Omron Sysmac Studio project Colorificio_grafica_MK.3 (Sysmac Studio 1.30.0.17, StandardProject)

# Controller PLC: NX1P2-9024DT1 version 1.40
Task PrimaryTask (priority 4, period or condition 2000): Program0
Library OmronLib_WC_Toolbox_V1_0 1.0.0 (contents left out)

TYPE S_Colori : STRUCT
    ALPHA : INT;
    RED : INT;
    GREEN : INT;
    BLU : INT;
    NOME : STRING[256];
END_STRUCT END_TYPE

VAR_GLOBAL
    SB0 : BOOL;  (* pulsante avvio ciclo automatico *)
    SB1 : BOOL;  (* pulsante arresto ciclo automatico *)
    SBE : BOOL;  (* pulsante arresto di emergenza *)
    YVA : BOOL;  (* libera caricatore seconda latta (A-) *)
    YVB : BOOL;  (* libera caricatore prima latta (B-) *)
    YVC : BOOL;  (* scarico bilancia (C+) *)
    KM1 : BOOL;  (* motore primo nastro *)
    KM2 : BOOL;  (* motore secondo nastro *)
    YVD : BOOL;  (* scarico coperchiatrice (D+) *)
    a0 : BOOL := False;  (* caricatore seconda latta libero (NA) *)
    a1 : BOOL := True;  (* caricatore seconda latta bloccato (NA) *)
    b0 : BOOL := False;  (* caricatore prima latta libero (NA) *)
    b1 : BOOL := True;  (* caricatore prima latta bloccato (NA) *)
    c0 : BOOL := True;  (* scaricatore bilancia rientrato (NA) *)
    c1 : BOOL := False;  (* scaricatore bilancia esteso (NA) *)
    d0 : BOOL := True;  (* scaricatore coperchiatrice rientrato (NA) *)
    d1 : BOOL := False;  (* scaricatore coperchiatrice esteso (NA) *)
    BIL : REAL;  (* bilancia/cella di carico (Grammi) *)
    YVBASE : BOOL;  (* eroga colorante base *)
    YVRED : BOOL;  (* eroga colorante rosso *)
    YVGREEN : BOOL;  (* eroga colorante verde *)
    YVBLU : BOOL;  (* eroga colorante blu *)
    YVSCARICO : BOOL;  (* eroga totale colore *)
    Tbase : TIME;  (* tempo carico base *)
    Trosso : TIME;  (* tempo carico rosso *)
    Tgreen : TIME;  (* tempo carico verde *)
    Tblu : TIME;  (* tempo carico blu *)
    BLW0 : BOOL := True;  (* livello minimo Base White (NA) *)
    BLW1 : BOOL := True;  (* livello riserva Base White (NA) *)
    BLR0 : BOOL := True;  (* livello minimo Red (NA) *)
    BLR1 : BOOL := True;  (* livello riserva Red (NA) *)
    BLG0 : BOOL := True;  (* livello minimo Green (NA) *)
    BLG1 : BOOL := True;  (* livello riserva Green (NA) *)
    BLB0 : BOOL := True;  (* livello minimo Blu (NA) *)
    BLB1 : BOOL := True;  (* livello riserva Blu (NA) *)
    BC0 : BOOL := False;  (* presenza prima latta sul caricatore (NA) *)
    BC1 : BOOL := False;  (* presenza seconda latta sul caricatore (NA) *)
    BBIL : BOOL := False;  (* presenza sulla bilancia (NA) *)
    BCOP : BOOL := False;  (* presenza sulla coperchiatrice (NA) *)
    ContattoValvolaBase : BOOL;
    ContattoValvolaRosso : BOOL;
    ContattoValvolaVerde : BOOL;
    ContattoValvolaBlu : BOOL;
    ContattoValvolaTramoggia : BOOL;
    LevelToEjectBase : INT := -1;
    LevelToEjectRosso : INT := -1;
    LevelToEjectVerde : INT := -1;
    LevelToEjectBlu : INT := -1;
    ColorDone : BOOL := False;
END_VAR

PROGRAM Program0
VAR
    TimerBase : TP;
    TimerRosso : TP;
    TimerVerde : TP;
    TimerBlu : TP;
    estimatedBase : TIME;
    estimatedRosso : TIME;
    estimatedVerde : TIME;
    estimatedBlu : TIME;
    SeqRGB : BOOL;
    Base : BOOL;
    Rosso : BOOL;
    Verde : BOOL;
    Blu : BOOL;
END_VAR
VAR_EXTERNAL
    SB1 : BOOL;
    KM1 : BOOL;
    YVC : BOOL;
    BBIL : BOOL;
    c0 : BOOL;
    c1 : BOOL;
    KM2 : BOOL;
    SB0 : BOOL;
    SBE : BOOL;
    BIL : REAL;
    ContattoValvolaBase : BOOL;
    ContattoValvolaRosso : BOOL;
    ContattoValvolaVerde : BOOL;
    ContattoValvolaBlu : BOOL;
    YVBASE : BOOL;
    YVRED : BOOL;
    YVGREEN : BOOL;
    YVBLU : BOOL;
    Tbase : TIME;
    Trosso : TIME;
    Tgreen : TIME;
    Tblu : TIME;
    ContattoValvolaTramoggia : BOOL;
    YVSCARICO : BOOL;
    LevelToEjectBase : INT;
    LevelToEjectRosso : INT;
    LevelToEjectVerde : INT;
    LevelToEjectBlu : INT;
    ColorDone : BOOL;  (* Finito il processo di carica della latta *)
END_VAR
VAR
    _p1 : BOOL;
    _p2 : BOOL;
    _p3 : BOOL;
END_VAR

(* Section Section0: ladder, written here as Structured Text *)

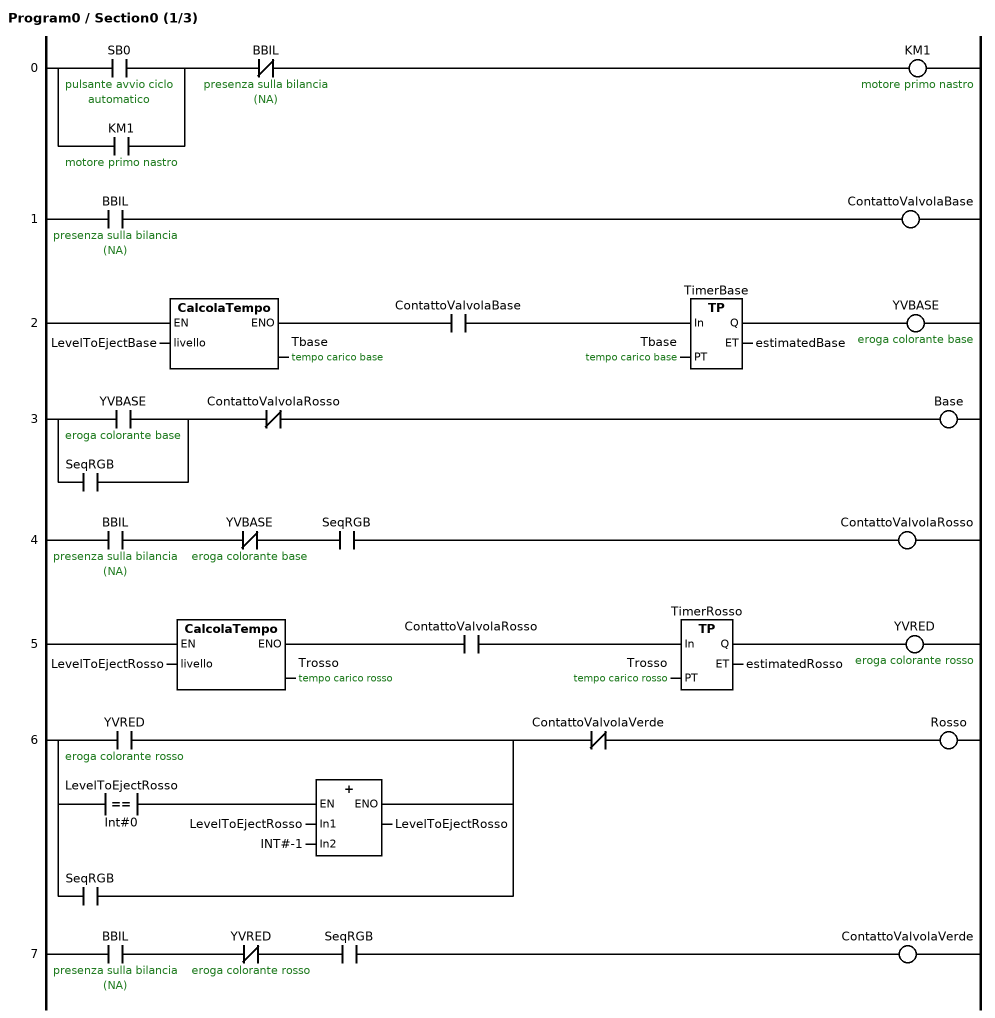
(* Rung 0 *)
KM1 := (SB0 OR KM1) AND NOT BBIL;
(* Rung 1 *)
ContattoValvolaBase := BBIL;
(* Rung 2 *)
Tbase := CalcolaTempo(livello := LevelToEjectBase);
TimerBase(In := ContattoValvolaBase, PT := Tbase, ET => estimatedBase);
YVBASE := TimerBase.Q;
(* Rung 3 *)
Base := (YVBASE OR SeqRGB) AND NOT ContattoValvolaRosso;
(* Rung 4 *)
ContattoValvolaRosso := BBIL AND NOT YVBASE AND SeqRGB;
(* Rung 5 *)
Trosso := CalcolaTempo(livello := LevelToEjectRosso);
TimerRosso(In := ContattoValvolaRosso, PT := Trosso, ET => estimatedRosso);
YVRED := TimerRosso.Q;
(* Rung 6 *)
_p1 := LevelToEjectRosso = Int#0;
IF _p1 THEN LevelToEjectRosso := LevelToEjectRosso + (INT#-1); END_IF;
Rosso := (YVRED OR _p1 OR SeqRGB) AND NOT ContattoValvolaVerde;
(* Rung 7 *)
ContattoValvolaVerde := BBIL AND NOT YVRED AND SeqRGB;

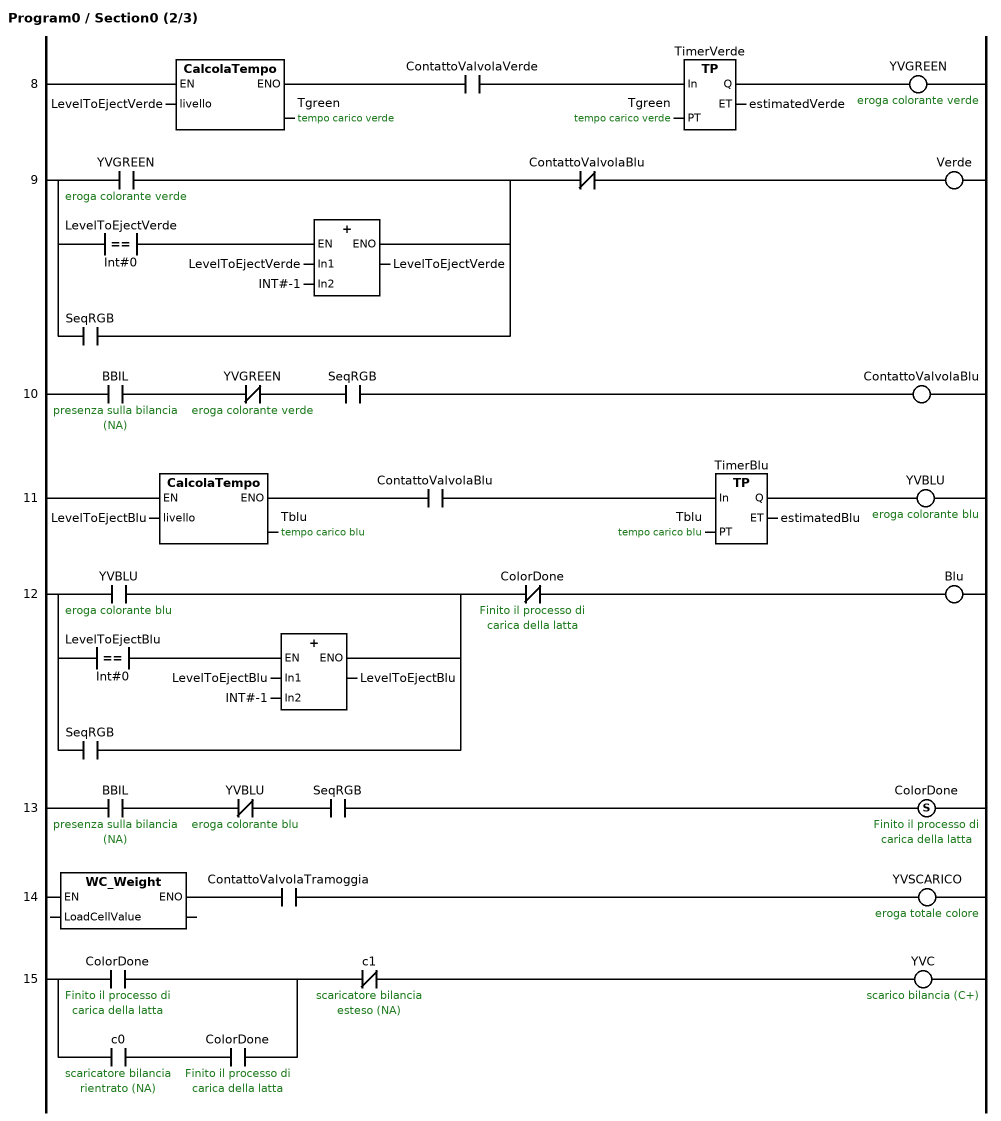
(* Rung 8 *)
Tgreen := CalcolaTempo(livello := LevelToEjectVerde);
TimerVerde(In := ContattoValvolaVerde, PT := Tgreen, ET => estimatedVerde);
YVGREEN := TimerVerde.Q;
(* Rung 9 *)
_p2 := LevelToEjectVerde = Int#0;
IF _p2 THEN LevelToEjectVerde := LevelToEjectVerde + (INT#-1); END_IF;
Verde := (YVGREEN OR _p2 OR SeqRGB) AND NOT ContattoValvolaBlu;
(* Rung 10 *)
ContattoValvolaBlu := BBIL AND NOT YVGREEN AND SeqRGB;
(* Rung 11 *)
Tblu := CalcolaTempo(livello := LevelToEjectBlu);
TimerBlu(In := ContattoValvolaBlu, PT := Tblu, ET => estimatedBlu);
YVBLU := TimerBlu.Q;
(* Rung 12 *)
_p3 := LevelToEjectBlu = Int#0;
IF _p3 THEN LevelToEjectBlu := LevelToEjectBlu + (INT#-1); END_IF;
Blu := (YVBLU OR _p3 OR SeqRGB) AND NOT ColorDone;
(* Rung 13 *)
IF BBIL AND NOT YVBLU AND SeqRGB THEN ColorDone := TRUE; END_IF;
(* Rung 14 *)
WC_Weight();
YVSCARICO := ContattoValvolaTramoggia;
(* Rung 15 *)
YVC := (ColorDone OR (c0 AND ColorDone)) AND NOT c1;

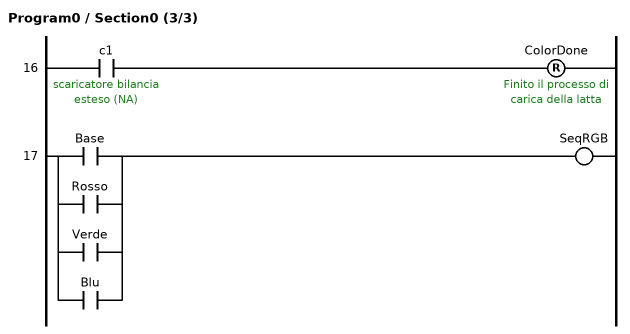
(* Rung 16 *)
IF c1 THEN ColorDone := FALSE; END_IF;
(* Rung 17 *)
SeqRGB := Base OR Rosso OR Verde OR Blu;
END_PROGRAM

FUNCTION WC_Weight : INT
VAR_INPUT
    LoadCellValue : INT;
END_VAR
// Il valore espresso è il peso in grammi
WC_Weight:=LoadCellValue*30; // LoadCellValue = livello colore della tramoggia di pesatura
END_FUNCTION

FUNCTION CalcolaTempo : TIME
VAR
    Temporanea : REAL;
END_VAR
VAR_INPUT
    livello : INT;
END_VAR
IF livello < 0 THEN
	CalcolaTempo := T#0s;
ELSE
	Temporanea := 0.2 ** 0.5; 
	Temporanea := Temporanea * 2 * livello;
	Temporanea := Temporanea ** 0.5;
	// Data la quantità di fluido da far uscire calcola il tempo che impiegherebbe supponendo che lo spazio da percorrere perchè il liquido superi la valvola sia di 20 cm = 0.2 m
	// Formula derivata dalla legge di Torricelli

	CalcolaTempo := NanoSecToTime(REAL_TO_INT(Temporanea) * 1000000000);
END_IF;
END_FUNCTION

# Device HMI (NA): not converted